// :Description: Filter state (library copy).
TYPE E_State :
(
    Idle := 0,
    Running := 1,
    Errored := 2
);
END_TYPE

(* stored: Version 1.1.0.1, ProductVersion 3.1.4026.0
   DUT E_State: Id {aaaaaaaa-aaaa-aaaa-aaaa-aaaaaaaaaaa3} *)
